# EPICS autosave request: tests/testfiles/cfg/SF_Mag_PV.req
$(SYS):ONOFF
$(SYS):I-SET
